(* PLC project MotionTest1, Higen MCL 1 *)
(* stored: creationDateTime 2012-01-06T15:20:13, modificationDateTime 2013-08-06T01:01:34 *)

FUNCTION_BLOCK PrepAxis
  VAR
    switch : MC_Power;
    readpos : MC_ReadActualPosition;
    readspeed : MC_ReadParameter;
  END_VAR
  VAR_INPUT
    Pwr : BOOL;
  END_VAR
  VAR
    MC_Sim1 : MC_Sim;
  END_VAR
  VAR_OUTPUT
    Axis : AXIS_REF;
    Position : LREAL;
    Velocity : LREAL;
  END_VAR

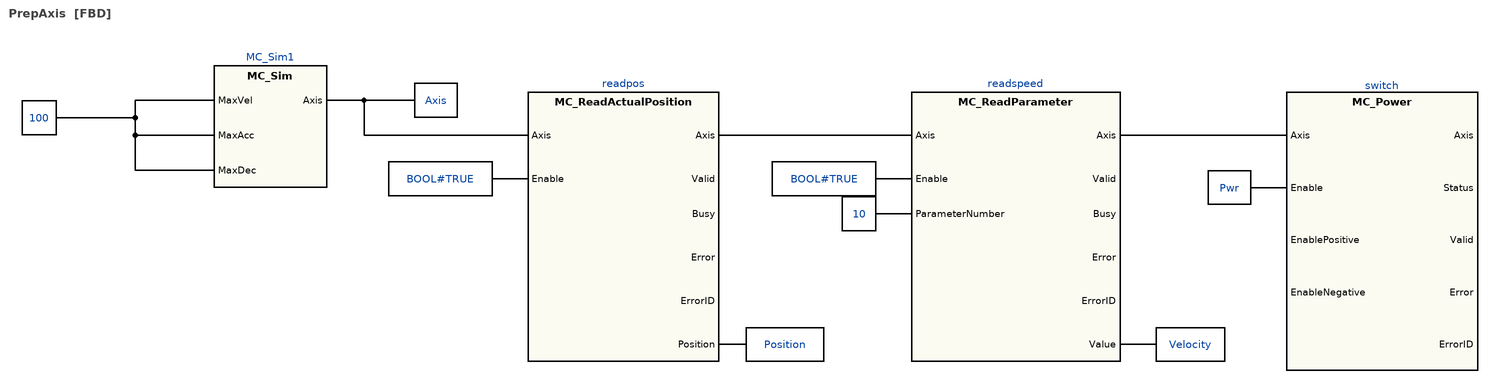
(* FBD diagram, written out as Structured Text *)
MC_Sim1(MaxVel := 100, MaxAcc := 100, MaxDec := 100);
Axis := MC_Sim1.Axis;
readpos(Axis := MC_Sim1.Axis, Enable := BOOL#TRUE);
Position := readpos.Position;
readspeed(Axis := readpos.Axis, Enable := BOOL#TRUE, ParameterNumber := 10);
Velocity := readspeed.Value;
switch(Axis := readspeed.Axis, Enable := Pwr);
END_FUNCTION_BLOCK

FUNCTION_BLOCK wxgetval
  VAR
    getpy : python_gear;
    latch : SR;
  END_VAR
  VAR_INPUT
    name : STRING;
  END_VAR
  VAR_OUTPUT
    val : BOOL;
  END_VAR
  VAR  (* added by the conversion: wires and edge detectors of the diagram *)
    _EQ41_ENO : BOOL;
    _EQ41_OUT : BOOL;
    _EQ3_ENO : BOOL;
    _EQ3_OUT : BOOL;
  END_VAR

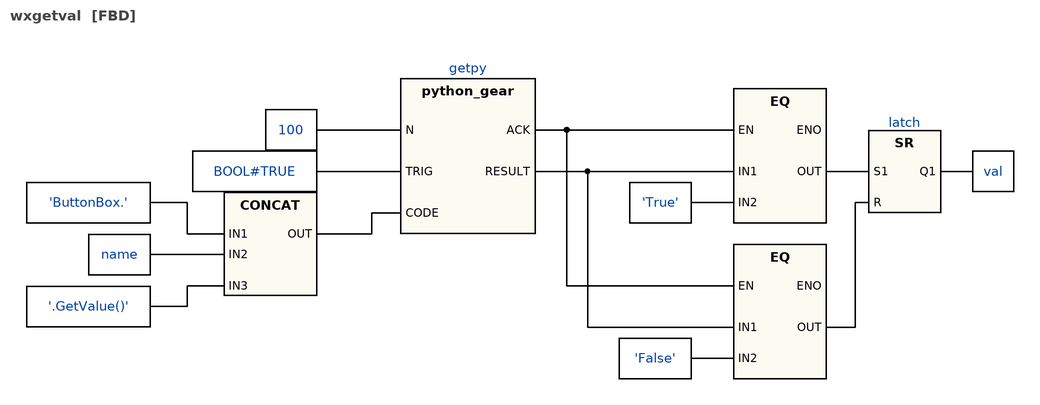
(* FBD diagram, written out as Structured Text *)
getpy(N := 100, TRIG := BOOL#TRUE, CODE := CONCAT('ButtonBox.', name, '.GetValue()'));
_EQ41_OUT := EQ(EN := getpy.ACK, IN1 := getpy.RESULT, IN2 := 'True', ENO => _EQ41_ENO);
_EQ3_OUT := EQ(EN := getpy.ACK, IN1 := getpy.RESULT, IN2 := 'False', ENO => _EQ3_ENO);
latch(S1 := _EQ41_OUT, R := _EQ3_OUT);
val := latch.Q1;
END_FUNCTION_BLOCK

(* - *)
PROGRAM main
  VAR
    MasterX : AXIS_REF;
    MasterY : AXIS_REF;
    MasterZ : AXIS_REF;
    MpX : LREAL;
    MpY : LREAL;
    MpZ : LREAL;
    MvX : LREAL;
    MvY : LREAL;
    MvZ : LREAL;
    SlaveX : AXIS_REF;
    SlaveY : AXIS_REF;
    SlaveZ : AXIS_REF;
    SpX : LREAL;
    SpY : LREAL;
    SpZ : LREAL;
    SvX : LREAL;
    SvY : LREAL;
    SvZ : LREAL;
  END_VAR
  VAR
    MasterKinTransform AT %IW1 : MC_KIN_REF;
    SlaveKinTransform AT %IW2 : MC_KIN_REF;
  END_VAR
  VAR
    bt1 : wxgetval;
    Block1 : wxgetval;
    Block2 : wxgetval;
    Block3 : wxgetval;
    Block6 : wxgetval;
    Block4 : wxgetval;
    Block7 : wxgetval;
    MC_IndexIdentInGroup0 : MC_IndexIdentInGroup;
    MC_AddAxisToGroup0 : MC_AddAxisToGroup;
    MC_CreateAxesGroup0 : MC_CreateAxesGroup;
    MC_AddAxisToGroup1 : MC_AddAxisToGroup;
    MC_IndexIdentInGroup1 : MC_IndexIdentInGroup;
    MC_GroupEnable0 : MC_GroupEnable;
    MC_AddAxisToGroup2 : MC_AddAxisToGroup;
    MC_IndexIdentInGroup2 : MC_IndexIdentInGroup;
    PrepAxis0 : PrepAxis;
    PrepAxis1 : PrepAxis;
    PrepAxis2 : PrepAxis;
    MasterGroup : AXES_GROUP_REF;
    SlaveGroup : AXES_GROUP_REF;
    MC_MoveDirectAbsolute0 : MC_MoveDirectAbsolute;
    MC_ToRealArray1 : MC_ToRealArray;
    MC_SetKinTransform0 : MC_SetKinTransform;
    PrepAxis3 : PrepAxis;
    PrepAxis4 : PrepAxis;
    PrepAxis5 : PrepAxis;
    MC_CreateAxesGroup1 : MC_CreateAxesGroup;
    MC_AddAxisToGroup3 : MC_AddAxisToGroup;
    MC_IndexIdentInGroup3 : MC_IndexIdentInGroup;
    MC_SetKinTransform1 : MC_SetKinTransform;
    MC_AddAxisToGroup4 : MC_AddAxisToGroup;
    MC_IndexIdentInGroup4 : MC_IndexIdentInGroup;
    MC_IndexIdentInGroup5 : MC_IndexIdentInGroup;
    MC_AddAxisToGroup5 : MC_AddAxisToGroup;
    MC_GroupEnable1 : MC_GroupEnable;
    MC_ToRealArray3 : MC_ToRealArray;
    MC_MoveDirectAbsolute1 : MC_MoveDirectAbsolute;
    MC_SetDynCoordTransform0 : MC_SetDynCoordTransform;
    MC_ToCoordinateTransform0 : MC_ToCoordinateTransform;
    MC_MoveLinearAbsolute0 : MC_MoveLinearAbsolute;
    MC_ToRealArray0 : MC_ToRealArray;
    MC_ToRealArray2 : MC_ToRealArray;
    MC_MoveLinearRelative0 : MC_MoveLinearRelative;
    MC_ToRealArray4 : MC_ToRealArray;
    MC_MoveLinearRelative1 : MC_MoveLinearRelative;
    MC_ToRealArray5 : MC_ToRealArray;
    MC_MoveLinearRelative2 : MC_MoveLinearRelative;
    MC_ToRealArray6 : MC_ToRealArray;
    MC_MoveLinearRelative3 : MC_MoveLinearRelative;
  END_VAR

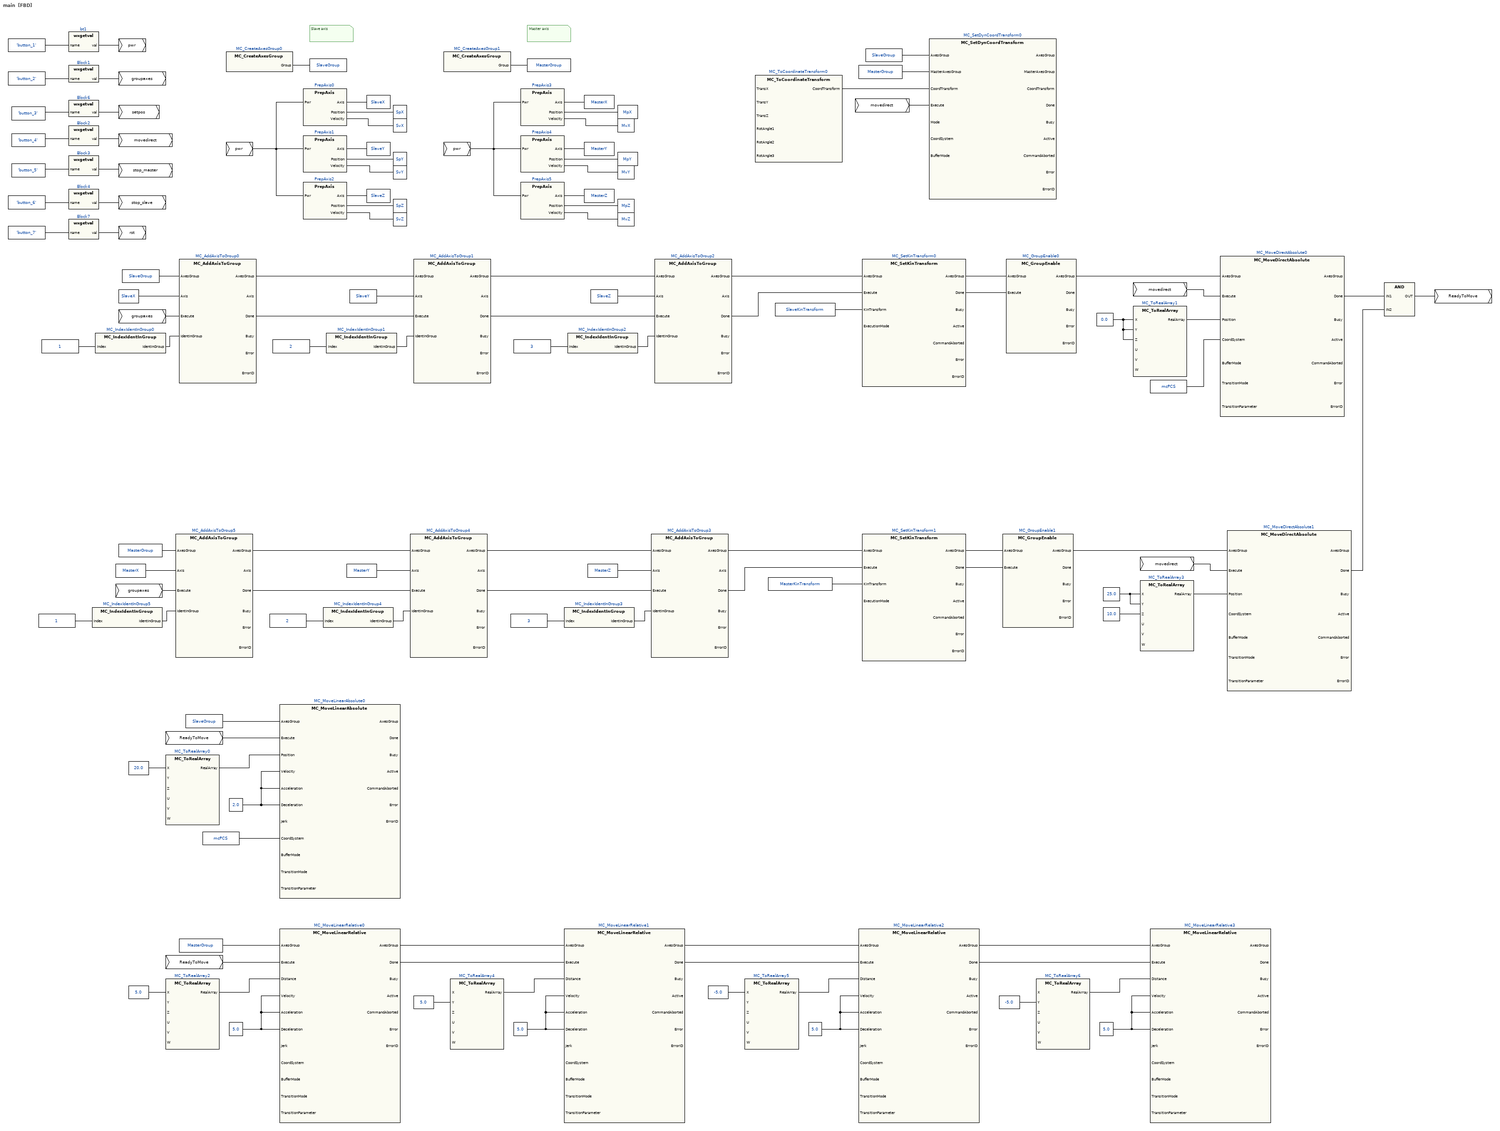
(* FBD diagram, written out as Structured Text *)
(* Slave axis *)
(* Master axis *)
MC_CreateAxesGroup0();
SlaveGroup := MC_CreateAxesGroup0.Group;
MC_CreateAxesGroup1();
MasterGroup := MC_CreateAxesGroup1.Group;
bt1(name := 'button_1');
PrepAxis0(Pwr := bt1.val);
SlaveX := PrepAxis0.Axis;
PrepAxis3(Pwr := bt1.val);
MasterX := PrepAxis3.Axis;
SpX := PrepAxis0.Position;
MpX := PrepAxis3.Position;
SvX := PrepAxis0.Velocity;
MvX := PrepAxis3.Velocity;
PrepAxis1(Pwr := bt1.val);
SlaveY := PrepAxis1.Axis;
PrepAxis4(Pwr := bt1.val);
MasterY := PrepAxis4.Axis;
SpY := PrepAxis1.Position;
MpY := PrepAxis4.Position;
SvY := PrepAxis1.Velocity;
MvY := PrepAxis4.Velocity;
PrepAxis2(Pwr := bt1.val);
SlaveZ := PrepAxis2.Axis;
PrepAxis5(Pwr := bt1.val);
MasterZ := PrepAxis5.Axis;
SpZ := PrepAxis2.Position;
MpZ := PrepAxis5.Position;
SvZ := PrepAxis2.Velocity;
MvZ := PrepAxis5.Velocity;
MC_ToCoordinateTransform0();
Block2(name := 'button_4');
MC_SetDynCoordTransform0(AxesGroup := SlaveGroup, MasterAxesGroup := MasterGroup, CoordTransform := MC_ToCoordinateTransform0.CoordTransform, Execute := Block2.val);
Block1(name := 'button_2');
Block6(name := 'button_3');
Block3(name := 'button_5');
Block4(name := 'button_6');
Block7(name := 'button_7');
MC_IndexIdentInGroup0(Index := 1);
MC_AddAxisToGroup0(AxesGroup := SlaveGroup, Axis := SlaveX, Execute := Block1.val, IdentInGroup := MC_IndexIdentInGroup0.IdentInGroup);
MC_IndexIdentInGroup1(Index := 2);
MC_AddAxisToGroup1(AxesGroup := MC_AddAxisToGroup0.AxesGroup, Axis := SlaveY, Execute := MC_AddAxisToGroup0.Done, IdentInGroup := MC_IndexIdentInGroup1.IdentInGroup);
MC_IndexIdentInGroup2(Index := 3);
MC_AddAxisToGroup2(AxesGroup := MC_AddAxisToGroup1.AxesGroup, Axis := SlaveZ, Execute := MC_AddAxisToGroup1.Done, IdentInGroup := MC_IndexIdentInGroup2.IdentInGroup);
MC_SetKinTransform0(AxesGroup := MC_AddAxisToGroup2.AxesGroup, Execute := MC_AddAxisToGroup2.Done, KinTransform := SlaveKinTransform);
MC_GroupEnable0(AxesGroup := MC_SetKinTransform0.AxesGroup, Execute := MC_SetKinTransform0.Done);
MC_ToRealArray1(X := 0.0, Y := 0.0, Z := 0.0);
MC_MoveDirectAbsolute0(AxesGroup := MC_GroupEnable0.AxesGroup, Execute := Block2.val, Position := MC_ToRealArray1.RealArray, CoordSystem := mcPCS);
MC_IndexIdentInGroup5(Index := 1);
MC_AddAxisToGroup5(AxesGroup := MasterGroup, Axis := MasterX, Execute := Block1.val, IdentInGroup := MC_IndexIdentInGroup5.IdentInGroup);
MC_IndexIdentInGroup4(Index := 2);
MC_AddAxisToGroup4(AxesGroup := MC_AddAxisToGroup5.AxesGroup, Axis := MasterY, Execute := MC_AddAxisToGroup5.Done, IdentInGroup := MC_IndexIdentInGroup4.IdentInGroup);
MC_IndexIdentInGroup3(Index := 3);
MC_AddAxisToGroup3(AxesGroup := MC_AddAxisToGroup4.AxesGroup, Axis := MasterZ, Execute := MC_AddAxisToGroup4.Done, IdentInGroup := MC_IndexIdentInGroup3.IdentInGroup);
MC_SetKinTransform1(AxesGroup := MC_AddAxisToGroup3.AxesGroup, Execute := MC_AddAxisToGroup3.Done, KinTransform := MasterKinTransform);
MC_GroupEnable1(AxesGroup := MC_SetKinTransform1.AxesGroup, Execute := MC_SetKinTransform1.Done);
MC_ToRealArray3(X := 25.0, Y := 25.0, Z := 10.0);
MC_MoveDirectAbsolute1(AxesGroup := MC_GroupEnable1.AxesGroup, Execute := Block2.val, Position := MC_ToRealArray3.RealArray);
MC_ToRealArray0(X := 20.0);
MC_MoveLinearAbsolute0(AxesGroup := SlaveGroup, Execute := MC_MoveDirectAbsolute0.Done AND MC_MoveDirectAbsolute1.Done, Position := MC_ToRealArray0.RealArray, Velocity := 2.0, Acceleration := 2.0, Deceleration := 2.0, CoordSystem := mcPCS);
MC_ToRealArray2(X := 5.0);
MC_MoveLinearRelative0(AxesGroup := MasterGroup, Execute := MC_MoveDirectAbsolute0.Done AND MC_MoveDirectAbsolute1.Done, Distance := MC_ToRealArray2.RealArray, Velocity := 5.0, Acceleration := 5.0, Deceleration := 5.0);
MC_ToRealArray4(Y := 5.0);
MC_MoveLinearRelative1(AxesGroup := MC_MoveLinearRelative0.AxesGroup, Execute := MC_MoveLinearRelative0.Done, Distance := MC_ToRealArray4.RealArray, Velocity := 5.0, Acceleration := 5.0, Deceleration := 5.0);
MC_ToRealArray5(X := -5.0);
MC_MoveLinearRelative2(AxesGroup := MC_MoveLinearRelative1.AxesGroup, Execute := MC_MoveLinearRelative1.Done, Distance := MC_ToRealArray5.RealArray, Velocity := 5.0, Acceleration := 5.0, Deceleration := 5.0);
MC_ToRealArray6(Y := -5.0);
MC_MoveLinearRelative3(AxesGroup := MC_MoveLinearRelative2.AxesGroup, Execute := MC_MoveLinearRelative2.Done, Distance := MC_ToRealArray6.RealArray, Velocity := 5.0, Acceleration := 5.0, Deceleration := 5.0);
END_PROGRAM

CONFIGURATION conf
  RESOURCE res ON PLC
    TASK milisecond(INTERVAL := T#10ms, PRIORITY := 0);
    PROGRAM maininstance WITH milisecond : main;
  END_RESOURCE
END_CONFIGURATION
